// Register function
FunctionRegistry[F_10_001_0227_01_0].Enable                            := TRUE; (* Function will be called *)
FunctionRegistry[F_10_001_0227_01_0].eFunctionNumber                   := fbF_10_001_0227_01_0.ConfigFunction.eFunctionNumber; // Registration number


(****************************** 10-001-0230-00-0 ************************************)
(*************************** ProBoxElement with one Motor *******************************)
// Configuration element 
fbEL_10_001_0230_00_0.ConfigElement.ElementName                     := '10-001-0230-00-0'; // Element name 
fbEL_10_001_0230_00_0.ConfigElement.eElementNumber                  := E_10_001_0230_00_0; // Number of the element 
fbEL_10_001_0230_00_0.ConfigElement.eSlaveElementNumber_34          := E_ElementNumber.E_BEGIN_ELEMENT; // Link from Master to slave element
fbEL_10_001_0230_00_0.ConfigElement.eElementType                    := E_ElementType.NO_TYPE; // No specific type

// Register element 
ElementRegistry[E_10_001_0230_00_0].Enable                          := TRUE; // Object is called
ElementRegistry[E_10_001_0230_00_0].eElementNumber                  := fbEL_10_001_0230_00_0.ConfigElement.eElementNumber; 

(****************************** 10-001-0230-01-0 ************************************)
(******************************** TransferCC  ***************************************)
// Configuration function
fbF_10_001_0230_01_0.ConfigFunction.FunctionName                      := '10-001-0230-01-0'; // Function name
fbF_10_001_0230_01_0.ConfigFunction.eFunctionNumber                   := F_10_001_0230_01_0; // Number of the function
fbF_10_001_0230_01_0.ConfigFunction.eElementLink                      := E_ElementNumber.E_10_001_0230_00_0;
fbF_10_001_0230_01_0.ConfigFunction.FunctionLink.eFunctionNumber      := E_FunctionNumber.F_BEGIN_FUNCTION;
fbF_10_001_0230_01_0.ConfigFunction.FunctionLink.ZoneNumber           := 0;
fbF_10_001_0230_01_0.ConfigFunction.eAdjacentFunctionNumberSide[1]    := E_FunctionNumber.F_10_001_0222_01_0;
fbF_10_001_0230_01_0.ConfigFunction.eAdjacentFunctionNumberSide[2]    := E_FunctionNumber.F_10_001_0232_01_0;
fbF_10_001_0230_01_0.ConfigFunction.eAdjacentFunctionNumberSide[3]    := E_FunctionNumber.F_BEGIN_FUNCTION;
fbF_10_001_0230_01_0.ConfigFunction.eAdjacentFunctionNumberSide[4]    := E_FunctionNumber.F_BEGIN_FUNCTION;
fbF_10_001_0230_01_0.ConfigFunction.ePrevFunctionNumber               := E_FunctionNumber.F_10_001_0222_01_0;
fbF_10_001_0230_01_0.ConfigFunction.eNextFunctionNumber               := E_FunctionNumber.F_BEGIN_FUNCTION;
fbF_10_001_0230_01_0.ConfigFunction.FlowDirectionREV                  := FALSE;
fbF_10_001_0230_01_0.ConfigFunction.NumberOfZones                     := 1;

fbF_10_001_0230_01_0.ConfigFunction.Zone[1].ZoneName                  := '10-001-0230-01-1';
fbF_10_001_0230_01_0.ConfigFunction.Zone[1].EnableMFC                 := TRUE;
fbF_10_001_0230_01_0.ConfigFunction.Zone[1].EnableLatchOccupiedState  := TRUE;
fbF_10_001_0230_01_0.ConfigFunction.Zone[1].Length[1]                 := 1400;


fbF_10_001_0230_01_0.Config.HomePosFree								  := E_Positions_HorizontalControl.LEFT;
fbF_10_001_0230_01_0.Config.HomePosOccupied							  := E_Positions_HorizontalControl.LEFT;
fbF_10_001_0230_01_0.Config.ReleaseBreakTime						  := T#500MS;
fbF_10_001_0230_01_0.Config.TimeoutValueMotor						  := T#30S;

// Register function
FunctionRegistry[F_10_001_0230_01_0].Enable                     		:= TRUE; (* Function will be called *)
FunctionRegistry[F_10_001_0230_01_0].eFunctionNumber 					:= fbF_10_001_0230_01_0.ConfigFunction.eFunctionNumber; // Registration number


(****************************** 10-001-0232-00-0 ************************************)
(*************************** ProBoxElement with one Motor *******************************)
// Configuration element 
fbEL_10_001_0232_00_0.ConfigElement.ElementName                     := '10-001-0232-00-0'; // Element name 
fbEL_10_001_0232_00_0.ConfigElement.eElementNumber                  := E_10_001_0232_00_0; // Number of the element 
fbEL_10_001_0232_00_0.ConfigElement.eSlaveElementNumber_34          := E_ElementNumber.E_BEGIN_ELEMENT; // Link from Master to slave element
fbEL_10_001_0232_00_0.ConfigElement.eElementType                    := E_ElementType.NO_TYPE; // No specific type

// Register element 
ElementRegistry[E_10_001_0232_00_0].Enable                          := TRUE; // Object is called
ElementRegistry[E_10_001_0232_00_0].eElementNumber                  := fbEL_10_001_0232_00_0.ConfigElement.eElementNumber; 

(****************************** 10-001-0232-01-0 ************************************)
(************************** ProBox Straight Transport *******************************)
// Configuration function
fbF_10_001_0232_01_0.ConfigFunction.FunctionName                       := '10-001-0232-01-0'; // Function name
fbF_10_001_0232_01_0.ConfigFunction.eFunctionNumber                    := F_10_001_0232_01_0; // Number of the function
fbF_10_001_0232_01_0.ConfigFunction.eElementLink                       := E_ElementNumber.E_10_001_0232_00_0;
fbF_10_001_0232_01_0.ConfigFunction.FunctionLink.eFunctionNumber       := E_FunctionNumber.F_BEGIN_FUNCTION;
fbF_10_001_0232_01_0.ConfigFunction.FunctionLink.ZoneNumber            := 0;
fbF_10_001_0232_01_0.ConfigFunction.eAdjacentFunctionNumberSide[1]     := E_FunctionNumber.F_10_001_0230_01_0;
fbF_10_001_0232_01_0.ConfigFunction.eAdjacentFunctionNumberSide[2]     := E_FunctionNumber.F_BEGIN_FUNCTION;
fbF_10_001_0232_01_0.ConfigFunction.ePrevFunctionNumber                := E_FunctionNumber.F_10_001_0230_01_0;
fbF_10_001_0232_01_0.ConfigFunction.eNextFunctionNumber                := E_FunctionNumber.F_BEGIN_FUNCTION;
fbF_10_001_0232_01_0.ConfigFunction.NumberOfZones                      := 2;
//Config zone 1
fbF_10_001_0232_01_0.ConfigFunction.Zone[1].ZoneName                   := '10-001-0232-01-1';
fbF_10_001_0232_01_0.ConfigFunction.Zone[1].EnableMFC                  := TRUE;
fbF_10_001_0232_01_0.ConfigFunction.Zone[1].EnableSimultaneousTransport:= TRUE; //Enable Simultaneous transport for multi zone functions
fbF_10_001_0232_01_0.ConfigFunction.Zone[1].EnableLatchOccupiedState   := TRUE;
fbF_10_001_0232_01_0.ConfigFunction.Zone[1].Length[1]                  := INT_TO_UINT(3000 / fbF_10_001_0232_01_0.ConfigFunction.NumberOfZones);	//Zone length (ie element length / number of zones)

//Config remaining zones equal to zone 1.
fbF_10_001_0232_01_0.ConfigFunction.Zone[2]                            := fbF_10_001_0232_01_0.ConfigFunction.Zone[1];
fbF_10_001_0232_01_0.ConfigFunction.Zone[2].ZoneName                   := '10-001-0232-01-2';

fbF_10_001_0232_01_0.Config.TwoSensorFunction                          := TRUE; // Slugging sensor present

// Register function
FunctionRegistry[F_10_001_0232_01_0].Enable                            := TRUE; (* Function will be called *)
FunctionRegistry[F_10_001_0232_01_0].eFunctionNumber                   := fbF_10_001_0232_01_0.ConfigFunction.eFunctionNumber; // Registration number


(****************************** 10-001-0232-02-0 ************************************)
(********************************* In/Out Feed ****************************************)
// Configuration function 
fbF_10_001_0232_02_0.ConfigFunction.FunctionName                     := '10-001-0232-02-0'; (* Function name *)
fbF_10_001_0232_02_0.ConfigFunction.eFunctionNumber                  := F_10_001_0232_02_0; (* Number of the function *)
fbF_10_001_0232_02_0.ConfigFunction.eElementLink                     := E_ElementNumber.E_10_001_0232_00_0; 
fbF_10_001_0232_02_0.ConfigFunction.FunctionLink.eFunctionNumber     := E_FunctionNumber.F_10_001_0232_01_0;	//Addon link to function, this is auto generated, an may need to be changed.
fbF_10_001_0232_02_0.ConfigFunction.FunctionLink.ZoneNumber          := 1;		

fbF_10_001_0232_02_0.Config.tFTLClearTime                  		  := T#5S; //Fork Truck Lift clear time
fbF_10_001_0232_02_0.Config.tTUSensorTime					  		  := T#5S; //Sensor occupied Time when to add or remove TU
fbF_10_001_0232_02_0.Config.TimeoutValueLift					  	  := T#10S; //Timeout value for lifting
fbF_10_001_0232_02_0.Config.LiftEnabled					  	  	  := FALSE; //Config if function has lift

// Register function 
FunctionRegistry[F_10_001_0232_02_0].Enable                           := TRUE; (* Function will be called *)
FunctionRegistry[F_10_001_0232_02_0].eFunctionNumber                  := fbF_10_001_0232_02_0.ConfigFunction.eFunctionNumber; (* Registration number *)


(****************************** 10-001-0233-00-0 ************************************)
(*************************** ProBoxElement with one Motor *******************************)
// Configuration element 
fbEL_10_001_0233_00_0.ConfigElement.ElementName                     := '10-001-0233-00-0'; // Element name 
fbEL_10_001_0233_00_0.ConfigElement.eElementNumber                  := E_10_001_0233_00_0; // Number of the element 
fbEL_10_001_0233_00_0.ConfigElement.eSlaveElementNumber_34          := E_ElementNumber.E_BEGIN_ELEMENT; // Link from Master to slave element
fbEL_10_001_0233_00_0.ConfigElement.eElementType                    := E_ElementType.NO_TYPE; // No specific type

// Register element 
ElementRegistry[E_10_001_0233_00_0].Enable                          := TRUE; // Object is called
ElementRegistry[E_10_001_0233_00_0].eElementNumber                  := fbEL_10_001_0233_00_0.ConfigElement.eElementNumber; 

(****************************** 10-001-0233-01-0 ************************************)
(************************** ProBox Straight Transport *******************************)
// Configuration function
fbF_10_001_0233_01_0.ConfigFunction.FunctionName                       := '10-001-0233-01-0'; // Function name
fbF_10_001_0233_01_0.ConfigFunction.eFunctionNumber                    := F_10_001_0233_01_0; // Number of the function
fbF_10_001_0233_01_0.ConfigFunction.eElementLink                       := E_ElementNumber.E_10_001_0233_00_0;
fbF_10_001_0233_01_0.ConfigFunction.FunctionLink.eFunctionNumber       := E_FunctionNumber.F_BEGIN_FUNCTION;
fbF_10_001_0233_01_0.ConfigFunction.FunctionLink.ZoneNumber            := 0;
fbF_10_001_0233_01_0.ConfigFunction.eAdjacentFunctionNumberSide[1]     := E_FunctionNumber.F_10_001_0204_01_0;
fbF_10_001_0233_01_0.ConfigFunction.eAdjacentFunctionNumberSide[2]     := E_FunctionNumber.F_BEGIN_FUNCTION;
fbF_10_001_0233_01_0.ConfigFunction.ePrevFunctionNumber                := E_FunctionNumber.F_10_001_0204_01_0;
fbF_10_001_0233_01_0.ConfigFunction.eNextFunctionNumber                := E_FunctionNumber.F_BEGIN_FUNCTION;
fbF_10_001_0233_01_0.ConfigFunction.NumberOfZones                      := 1;
//Config zone 1
fbF_10_001_0233_01_0.ConfigFunction.Zone[1].ZoneName                   := '10-001-0233-01-1';
fbF_10_001_0233_01_0.ConfigFunction.Zone[1].EnableMFC                  := TRUE;
fbF_10_001_0233_01_0.ConfigFunction.Zone[1].EnableSimultaneousTransport:= FALSE; //Disable Simultaneous transport for multi zone functions
fbF_10_001_0233_01_0.ConfigFunction.Zone[1].EnableLatchOccupiedState   := TRUE;
fbF_10_001_0233_01_0.ConfigFunction.Zone[1].Length[1]                  := INT_TO_UINT(1600 / fbF_10_001_0233_01_0.ConfigFunction.NumberOfZones);	//Zone length (ie element length / number of zones)

// Register function
FunctionRegistry[F_10_001_0233_01_0].Enable                            := TRUE; (* Function will be called *)
FunctionRegistry[F_10_001_0233_01_0].eFunctionNumber                   := fbF_10_001_0233_01_0.ConfigFunction.eFunctionNumber; // Registration number

END_FUNCTION

(* stored: Version 1.1.0.1, ProductVersion 3.1.4024.9
   POU F_ConfigPosition_001: Id {984f4fe4-d68f-4109-b494-91c37032a7d9}, SpecialFunc None *)
